TYPE "UDT without sub udt"
TITLE = has no title
VERSION : 0.1
//some comment
   STRUCT
      one : Bool;   // comment one
      two : Byte;   // comment two
      three : Word;   // comment three
      four : DWord;   // comment four
      five : LWord;   // comment five
      six : SInt;   // comment six
      seven : USInt;   // comment seven
      eight : Int;   // comment eight
      nine : UInt;   // comment nine
      ten : DInt;   // comment ten
      eleven : UDInt;   // comment eleven
      twelve : LInt;   // comment twelve
      thirteen : ULInt;   // comment thirteen
      fourteen : Real;   // comment fourteen
      fifteen : LReal;   // comment fifteen
      sixteen : Char;   // comment sixteen
      seventeen : WChar;   // comment seventeen
      eighteen : String;   // comment eighteen
      nineteen : WString;   // comment nineteen
      twenty {InstructionName := 'DTL'; LibVersion := '1.0'} : DTL;   // comment twenty
      twentyone : Array[0..10] of Byte;   // comment twentyone
      twentytwo : Struct   // comment twentytwo
         one : Bool;   // comment one
         two : Int;   // comment  two
         three : DInt;   // comment three
      END_STRUCT;
   END_STRUCT;

END_TYPE

